// TwinCAT 3 PLC project Main_project
// ProgramVersion: 3.1.4023.0
// libraries:
//   Tc2_Standard, * (Beckhoff Automation GmbH)
//   Tc2_System, * (Beckhoff Automation GmbH)
//   Tc3_Module, * (Beckhoff Automation GmbH)
// project tree:
//   GVLs/ GVL.TcGVL
//   / PlcTask.TcTTO
//   POUs/Devices/ Contactor.TcPOU, DirectOnlineStarterMotor.TcPOU, I_PushButton.TcIO, I_Sensor.TcIO, I_SingleDirectionMotor.TcIO, NormallyClosedSensor.TcPOU, NormallyOpenPushButton.TcPOU, NormallyClosedPushButton.TcPOU, NormallyOpenSensor.TcPOU
//   POUs/Machine/ MyConveyorSortingMachine.TcPOU
//   POUs/ MAIN.TcPOU
//   POUs/Module/ I_Module.TcIO, SortingConveyor.TcPOU
// real-time tasks:
//   TASK PlcTask: cycle T#10ms, priority 20, ADS port 350

CONFIGURATION Main_project
    RESOURCE PLC ON TwinCAT3
        TASK PlcTask(INTERVAL := T#10ms, PRIORITY := 20);
        PROGRAM MAIN WITH PlcTask : MAIN;
    END_RESOURCE
END_CONFIGURATION

// ---- GVLs/GVL.TcGVL
{attribute 'qualified_only'}
VAR_GLOBAL
	startButton	:	NormallyOpenPushButton;
	stopButton	:	NormallyClosedPushButton;
	emergencyStopButton	:	NormallyClosedPushButton;
	productDetectedSensor	:	NormallyClosedSensor;
	conveyorFullSensor	:	NormallyClosedSensor;
	conveyorMotor	:	DirectOnlineStarterMotor;
	
	sortingConveyor	:	SortingConveyor(ProductDetected := productDetectedSensor,
		                                ConveyorFull := conveyorFullSensor,
										ConveyorMotor := conveyorMotor);
	
	myConveyorSortingMachine	:	MyConveyorSortingMachine( StartButton := startButton,
                                                              StopButton := stopButton,
															  EmergencyStopButton := emergencyStopButton,
															  ConveyorModule := sortingConveyor);
END_VAR

// ---- POUs/Devices/I_PushButton.TcIO
INTERFACE I_PushButton

PROPERTY IsPressed : BOOL
GET
END_GET
END_PROPERTY

PROPERTY PUBLIC IsReleased : BOOL
GET
END_GET
END_PROPERTY

END_INTERFACE

// ---- POUs/Devices/I_Sensor.TcIO
INTERFACE I_Sensor

PROPERTY PUBLIC IsActive : BOOL
GET
END_GET
END_PROPERTY

END_INTERFACE

// ---- POUs/Devices/I_SingleDirectionMotor.TcIO
INTERFACE I_SingleDirectionMotor

METHOD PUBLIC Start
VAR_INPUT
END_VAR
END_METHOD

METHOD PUBLIC Stop
VAR_INPUT
END_VAR
END_METHOD

END_INTERFACE

// ---- POUs/Module/I_Module.TcIO
INTERFACE I_Module

METHOD Disable
VAR_INPUT
END_VAR
END_METHOD

METHOD Enable
VAR_INPUT
END_VAR
END_METHOD

END_INTERFACE

// ---- POUs/MAIN.TcPOU
PROGRAM MAIN
VAR
	ConveyorControl	:	BOOL;
	Timeout	:	TOF;
END_VAR

GVL.myConveyorSortingMachine();

Timeout(In := ConveyorControl AND GVL.ProductDetectedSensor.IsActive, PT := T#5S);

IF ConveyorControl AND Timeout.Q AND NOT GVL.ConveyorFullSensor.IsActive THEN
	GVL.ConveyorMotor.Start();
ELSE
	GVL.ConveyorMotor.Stop();
END_IF

END_PROGRAM

// ---- POUs/Machine/MyConveyorSortingMachine.TcPOU
FUNCTION_BLOCK MyConveyorSortingMachine
VAR
	_StartButton	:	I_PushButton;
	_StopButton	:	I_PushButton;
	_EmergencyStopButton	:	I_PushButton;
	_ConveyorModule	:	I_Module;
END_VAR

IF _StopButton.IsPressed OR _EmergencyStopButton.IsPressed THEN
	
	_ConveyorModule.Disable();
	
ELSIF _StartButton.IsPressed AND _StopButton.IsReleased AND _EmergencyStopButton.IsReleased THEN
	
	_ConveyorModule.Enable();
	
END_IF

METHOD FB_init : BOOL
VAR_INPUT
	bInitRetains :	BOOL; // if TRUE, the retain variables are initialized (warm start / cold start)
	bInCopyCode :	BOOL;  // if TRUE, the instance afterwards gets moved into the copy code (online change)
	StartButton	:	I_PushButton;
	StopButton	:	I_PushButton;
	EmergencyStopButton	:	I_PushButton;
	ConveyorModule	:	I_Module;

END_VAR
// ATTENZIONE ALLO scope delle variabili !!
// usare THIS^ per dereferenziare le variabili locali 
// di questa istanza della classe MyConveyorSortingMachine
THIS^._StartButton := StartButton;
THIS^._StopButton := StopButton;
THIS^._EmergencyStopButton := EmergencyStopButton;
THIS^._ConveyorModule := ConveyorModule;
END_METHOD

END_FUNCTION_BLOCK

// ---- POUs/Devices/NormallyOpenPushButton.TcPOU
FUNCTION_BLOCK NormallyOpenPushButton IMPLEMENTS I_PushButton
VAR
	input AT %I*	:	BOOL;
END_VAR

PROPERTY PUBLIC IsPressed : BOOL

// ho eliminato manualmente il Setter di questa proprietà perché qui non ha senso
GET
IsPressed := input;
END_GET
END_PROPERTY

PROPERTY PUBLIC IsReleased : BOOL

// ho eliminato manualmente il Setter di questa proprietà perché qui non ha senso
GET
IsReleased := NOT IsPressed;
END_GET
END_PROPERTY

END_FUNCTION_BLOCK

// ---- POUs/Devices/NormallyClosedPushButton.TcPOU
FUNCTION_BLOCK NormallyClosedPushButton IMPLEMENTS I_PushButton
VAR
	input AT %I*	:	BOOL;
END_VAR

PROPERTY PUBLIC IsPressed : BOOL

// ho eliminato manualmente il Setter di questa proprietà perché qui non ha senso
GET
IsPressed := NOT input;
END_GET
END_PROPERTY

PROPERTY PUBLIC IsReleased : BOOL

// ho eliminato manualmente il Setter di questa proprietà perché qui non ha senso
GET
IsReleased := NOT IsPressed;
END_GET
END_PROPERTY

END_FUNCTION_BLOCK

// ---- POUs/Devices/NormallyClosedSensor.TcPOU
FUNCTION_BLOCK NormallyClosedSensor IMPLEMENTS I_Sensor
VAR
	input AT %I*	:	BOOL;
END_VAR

PROPERTY PUBLIC IsActive : BOOL

// ho eliminato manualmente il Setter di questa proprietà perché qui non ha senso
GET
IsActive := NOT input;
END_GET
END_PROPERTY

END_FUNCTION_BLOCK

// ---- POUs/Devices/DirectOnlineStarterMotor.TcPOU
FUNCTION_BLOCK DirectOnlineStarterMotor implements I_SingleDirectionMotor
VAR
	contactor	:	Contactor;
END_VAR

METHOD PUBLIC Start
VAR_INPUT
END_VAR
contactor.SwitchOn();
END_METHOD

METHOD PUBLIC Stop
VAR_INPUT
END_VAR
contactor.SwitchOff();
END_METHOD

END_FUNCTION_BLOCK

// ---- POUs/Devices/Contactor.TcPOU
FUNCTION_BLOCK Contactor
VAR
	output AT %Q*	:	BOOL;
END_VAR

METHOD PUBLIC SwitchOff
VAR_INPUT
END_VAR
output := FALSE;
END_METHOD

METHOD PUBLIC SwitchOn
VAR_INPUT
END_VAR
output := TRUE;
END_METHOD

END_FUNCTION_BLOCK

// ---- POUs/Module/SortingConveyor.TcPOU
FUNCTION_BLOCK SortingConveyor IMPLEMENTS I_Module
VAR
	_productDetected	:	I_Sensor;
	_conveyorFull	:	I_Sensor;
	_conveyorMotor	:	I_SingleDirectionMotor;
	_enabled	:	BOOL;
	_timeout: TOF;
END_VAR

_timeout(In := _enabled AND _productDetected.IsActive, PT := T#5S);

IF _enabled AND _timeout.Q AND NOT _conveyorFull.IsActive THEN
	_conveyorMotor.Start();
ELSE
	_conveyorMotor.Stop();
END_IF

METHOD Disable
VAR_INPUT
END_VAR
_enabled := false;
END_METHOD

METHOD Enable
VAR_INPUT
END_VAR
_enabled := true;
END_METHOD

METHOD FB_init : BOOL
VAR_INPUT
	bInitRetains : BOOL; // if TRUE, the retain variables are initialized (warm start / cold start)
	bInCopyCode : BOOL;  // if TRUE, the instance afterwards gets moved into the copy code (online change)
	ProductDetected	:	I_Sensor;
	ConveyorFull	:	I_Sensor;
	ConveyorMotor	:	I_SingleDirectionMotor;
END_VAR
// ATTENZIONE ALLO scope delle variabili !!
// usare THIS^ per dereferenziare le variabili locali 
// di questa istanza della classe SortingConveyor
THIS^._productDetected := ProductDetected;
THIS^._conveyorFull := ConveyorFull;
this^._conveyorMotor := ConveyorMotor;
END_METHOD

END_FUNCTION_BLOCK

// ---- POUs/Devices/NormallyOpenSensor.TcPOU
FUNCTION_BLOCK NormallyOpenSensor IMPLEMENTS I_Sensor
VAR
	input AT %I*	:	BOOL;
END_VAR

PROPERTY PUBLIC IsActive : BOOL

// ho eliminato manualmente il Setter di questa proprietà perché qui non ha senso
GET
IsActive := input;
END_GET
END_PROPERTY

END_FUNCTION_BLOCK
